% RSLogix 500 project PROJECT5_DIGITAL_ROTAMETER.RSS, saved by version 8.30.00.16 %
PROJECT "UNTITLED"    % processor: Bul.1763 MicroLogix 1100 Series B %

PROGRAM FILES
  LAD 2 "MAIN"  7 rungs

DATA FILES
  O0 OUTPUT  4 elements
  I1 INPUT  6 elements
  S2 STATUS  66 elements
  B3 BINARY  1 elements
  T4 TIMER  1 elements
  C5 COUNTER  1 elements
  R6 CONTROL  1 elements
  N7 INTEGER  1 elements
  F8 FLOAT  1 elements

LADDER 2 "MAIN"
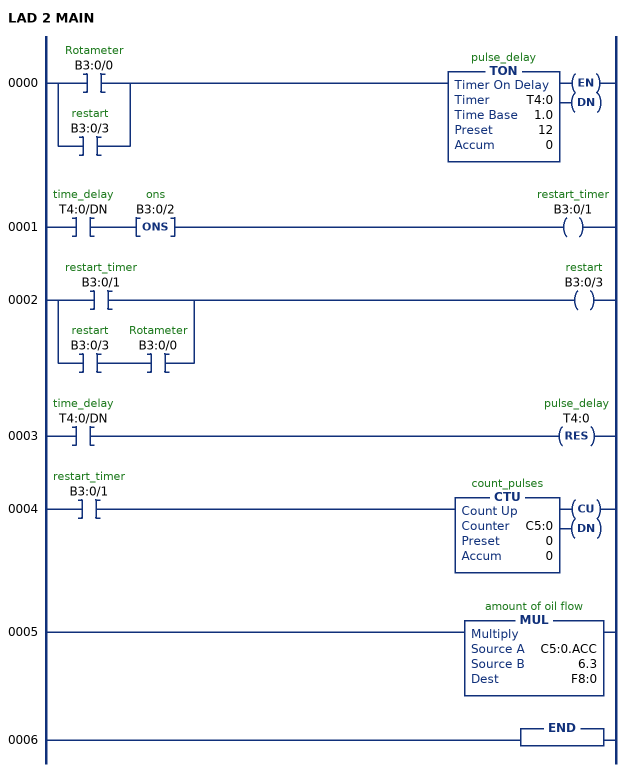
% Rung: 0 %
SOR BST XIC B3:0/0 NXB XIC B3:0/3 BND TON T4:0 1.0 12 0 EOR
%   B3:0/0  "Rotameter" %
%   B3:0/3  "restart" %
%   T4:0  "pulse_delay" %
% Rung: 1 %
SOR XIC T4:0/DN ONS B3:0/2 OTE B3:0/1 EOR
%   T4:0/DN  "time_delay" %
%   B3:0/2  "ons" %
%   B3:0/1  "restart_timer" %
% Rung: 2 %
SOR BST XIC B3:0/1 NXB XIC B3:0/3 XIC B3:0/0 BND OTE B3:0/3 EOR
%   B3:0/1  "restart_timer" %
%   B3:0/3  "restart" %
%   B3:0/0  "Rotameter" %
% Rung: 3 %
SOR XIC T4:0/DN RES T4:0 EOR
%   T4:0/DN  "time_delay" %
%   T4:0  "pulse_delay" %
% Rung: 4 %
SOR XIC B3:0/1 CTU C5:0 0 0 EOR
%   B3:0/1  "restart_timer" %
%   C5:0  "count_pulses" %
% Rung: 5 %
SOR MUL C5:0.ACC 6.3 F8:0 EOR
%   C5:0.ACC  "pulser" %
%   F8:0  "amount of oil flow" %
% Rung: 6 %
SOR END EOR

DATA TABLE (non-zero values as saved)
DATA T4
% .PRE .ACC %
% T4:0 % 12 0
